INTERFACE ITF_Group1_HMI_Init EXTENDS ITF_BaseGroupElement, ITF_Group1_HMI_Connector

END_INTERFACE

(* stored: Version 1.1.0.1
   Itf ITF_Group1_HMI_Init: Id {c1fd176f-5b4e-0bd8-0a85-b6edd03fbd79} *)
